// SIMATIC S7-200 SMART project (STEP 7-Micro/WIN SMART), CPU SR30

SYMBOL_TABLE 表格 1
控制发送             V162.0
END_SYMBOL_TABLE

SYMBOL_TABLE 系统符号
自动发生接通           V32.0
First_Scan_On    SM0.1    // 仅在第一个扫描周期时接通
END_SYMBOL_TABLE

ORGANIZATION_BLOCK 程序块:OB1
TITLE=
BEGIN
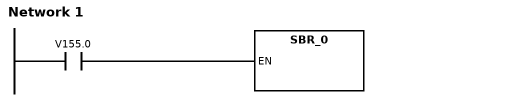
Network 1
LD     V155.0
CALL   SBR_0:SBR0
END_ORGANIZATION_BLOCK

SUBROUTINE_BLOCK SBR_0:SBR0
TITLE=干燥部分程序
BEGIN
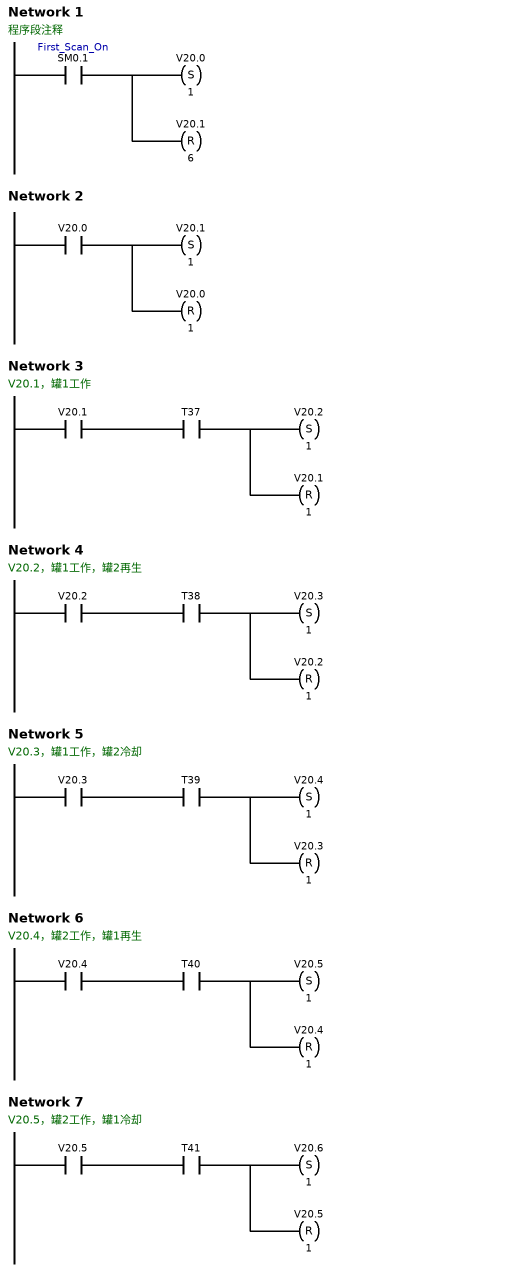
Network 1
// 程序段注释
LD     First_Scan_On:SM0.1
S      V20.0, 1
R      V20.1, 6
Network 2
LD     V20.0
S      V20.1, 1
R      V20.0, 1
Network 3
// V20.1，罐1工作
LD     V20.1
A      T37
S      V20.2, 1
R      V20.1, 1
Network 4
// V20.2，罐1工作，罐2再生
LD     V20.2
A      T38
S      V20.3, 1
R      V20.2, 1
Network 5
// V20.3，罐1工作，罐2冷却
LD     V20.3
A      T39
S      V20.4, 1
R      V20.3, 1
Network 6
// V20.4，罐2工作，罐1再生
LD     V20.4
A      T40
S      V20.5, 1
R      V20.4, 1
Network 7
// V20.5，罐2工作，罐1冷却
LD     V20.5
A      T41
S      V20.6, 1
R      V20.5, 1
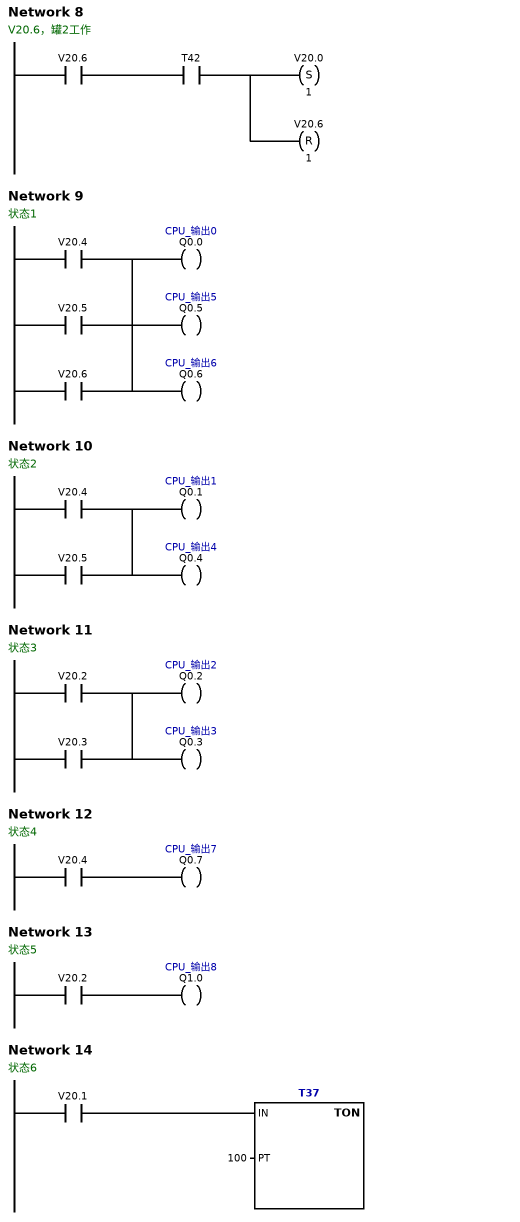
Network 8
// V20.6，罐2工作
LD     V20.6
A      T42
S      V20.0, 1
R      V20.6, 1
Network 9
// 状态1
LD     V20.4
O      V20.5
O      V20.6
=      CPU_输出0:Q0.0
=      CPU_输出5:Q0.5
=      CPU_输出6:Q0.6
Network 10
// 状态2
LD     V20.4
O      V20.5
=      CPU_输出1:Q0.1
=      CPU_输出4:Q0.4
Network 11
// 状态3
LD     V20.2
O      V20.3
=      CPU_输出2:Q0.2
=      CPU_输出3:Q0.3
Network 12
// 状态4
LD     V20.4
=      CPU_输出7:Q0.7
Network 13
// 状态5
LD     V20.2
=      CPU_输出8:Q1.0
Network 14
// 状态6
LD     V20.1
TON    T37, 100
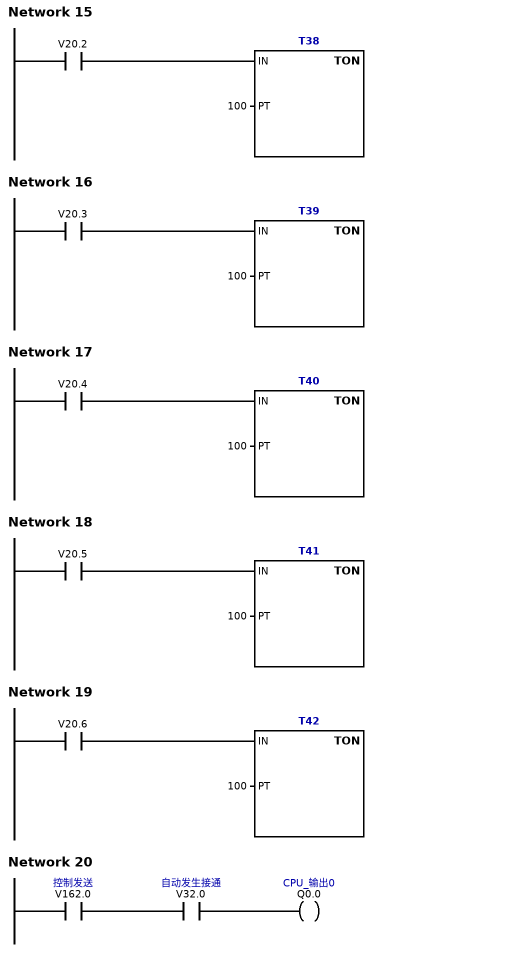
Network 15
LD     V20.2
TON    T38, 100
Network 16
LD     V20.3
TON    T39, 100
Network 17
LD     V20.4
TON    T40, 100
Network 18
LD     V20.5
TON    T41, 100
Network 19
LD     V20.6
TON    T42, 100
Network 20
LD     控制发送:V162.0
A      自动发生接通:V32.0
=      CPU_输出0:Q0.0
Network 26
// 程序段注释
END_SUBROUTINE_BLOCK
